// TIA Portal V17 export
// export: Created 2025-03-10T12:18:54.0403553Z, ExportSetting WithDefaults, DisplayName Totally Integrated Automation Portal, DisplayVersion V17 Update 8, DisplayName TIA Portal Openness, DisplayVersion V17 Update 8, DisplayName TIA Portal Version Control Interface, DisplayVersion V17, DisplayName SINAMICS Startdrive Advanced, DisplayVersion V17 SP2, DisplayName SINAMICS Startdrive G110M, G120, G120C, G120D, G120P, G115D, DisplayVersion V17 SP2, DisplayName SINAMICS Startdrive G130, G150, S120, S150, SINAMICS MV, S210, DisplayVersion V17 SP2, DisplayName STEP 7 Professional, DisplayVersion V17 Update 8, DisplayName SINUMERIK ONE STEP 7 Toolbox, DisplayVersion V17 Update 12, DisplayName SINUMERIK 840D sl STEP 7 Toolbox, DisplayVersion V17 Update 12, DisplayName STEP 7 Safety, DisplayVersion V17 Update 6, DisplayName WinCC Advanced, DisplayVersion V17 Update 8
FUNCTION_BLOCK "FB22107_WP321_MUL_CALL"   // FB22107, LAD
{ S7_Optimized_Access := 'FALSE' }
VERSION : 0.1
// stored: AutoNumber false, IsIECCheckEnabled false, SetENOAutomatically false, UDAEnableTagReadback false
   VAR_INPUT
      SynchronizeAllDataFromSiwarexToDataBlockOnStartUp : Bool;
   END_VAR
   VAR_OUTPUT
      ArrayStartValue : Int;
      ArrayMaxValue : Int;
   END_VAR
   VAR
      WP321DR { S7_SetPoint := 'True'} : Array[#ArrayStart..#ArrayLenghtMax] of "WP321DR";
   END_VAR
   VAR DB_SPECIFIC
      FBStartUpTemp { S7_SetPoint := 'True'} : Array[#ArrayStart..#ArrayLenghtMax] of Bool;
   END_VAR
   VAR_TEMP
      loop_count : Int;
   END_VAR
   VAR CONSTANT
      ArrayStart : Int;
      ArrayLenghtMax : Int := 7;
   END_VAR
   // WP321DR[0].HW_ID := 443;
   // WP321DR[1].HW_ID := 444;
   // WP321DR[2].HW_ID := 445;
   // WP321DR[3].HW_ID := 446;
   // WP321DR[4].HW_ID := 447;
   // WP321DR[5].HW_ID := 448;
   // WP321DR[6].HW_ID := 449;
   // WP321DR[7].HW_ID := 442;
   VAR_TEMP   // added for the SCL form of the ladder/FBD networks
      _w1 : Bool;
   END_VAR
BEGIN

REGION Network 1: Initializing of array pointers for loop
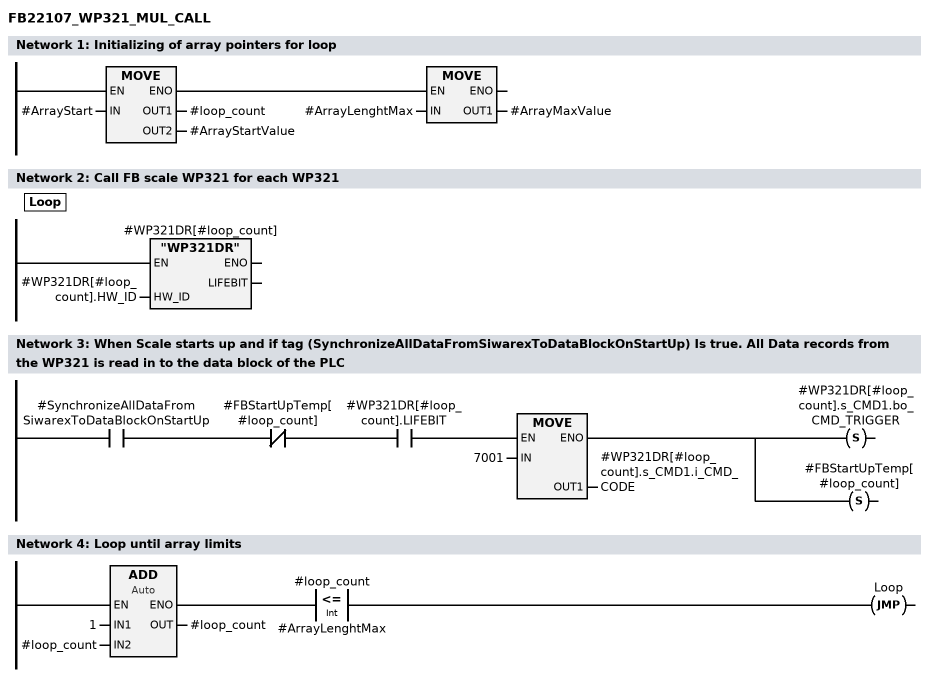
   RUNG wire#powerrail
      Move(in := #ArrayStart, out1 => #loop_count, out2 => #ArrayStartValue)
      Move(in := #ArrayLenghtMax, out1 => #ArrayMaxValue)
   END_RUNG
   // the same network as SCL:
   #loop_count := #ArrayStart;
   #ArrayStartValue := #ArrayStart;
   #ArrayMaxValue := #ArrayLenghtMax;
END_REGION

REGION Network 2: Call FB scale WP321 for each WP321
   Label( Loop )
   RUNG wire#powerrail
      #WP321DR[#loop_count](HW_ID := #WP321DR[#loop_count].HW_ID, LIFEBIT =>)
   END_RUNG
   // the same network as SCL:
   Loop:
   #WP321DR[#loop_count](HW_ID := #WP321DR[#loop_count].HW_ID);   // "WP321DR"
END_REGION

REGION Network 3: When Scale starts up and if tag (SynchronizeAllDataFromSiwarexToDataBlockOnStartUp) Is true. All Data records from the WP321 is read in to the data block of the PLC
   RUNG wire#powerrail
      Contact( #SynchronizeAllDataFromSiwarexToDataBlockOnStartUp )
      I_Contact( #FBStartUpTemp[#loop_count] )
      Contact( #WP321DR[#loop_count].LIFEBIT )
      Move(in := 7001, out1 => #WP321DR[#loop_count].s_CMD1.i_CMD_CODE)
      wire#w1
      S_Coil( #WP321DR[#loop_count].s_CMD1.bo_CMD_TRIGGER )
   END_RUNG
   RUNG wire#w1
      S_Coil( #FBStartUpTemp[#loop_count] )
   END_RUNG
   // the same network as SCL:
   #_w1 := #SynchronizeAllDataFromSiwarexToDataBlockOnStartUp AND NOT #FBStartUpTemp[#loop_count] AND #WP321DR[#loop_count].LIFEBIT;
   IF #_w1 THEN
       #WP321DR[#loop_count].s_CMD1.i_CMD_CODE := 7001;
       #WP321DR[#loop_count].s_CMD1.bo_CMD_TRIGGER := TRUE;
       #FBStartUpTemp[#loop_count] := TRUE;
   END_IF;
END_REGION

REGION Network 4: Loop until array limits
   RUNG wire#powerrail
      Add(in1 := 1, in2 := #loop_count, out => #loop_count)
      { S7_Templates := "SrcType := Int" } LE_Contact(in1 := #loop_count, in2 := #ArrayLenghtMax)
      JumpCoil( Loop )
   END_RUNG
   // the same network as SCL:
   #loop_count := 1 + #loop_count;
   IF #loop_count <= #ArrayLenghtMax THEN GOTO Loop; END_IF;
END_REGION
END_FUNCTION_BLOCK
